FUNCTION_BLOCK TLController (* Composite Function Block Type *)
  (* Standard: 61499-2 *)
  (* Version 0.2, 2003-12-05, JHC, Rockwell Automation, Renamed from NEWCOMPFB. *)
  (* Version 0.1, 2002-01-08, JHC, Rockwell Automation, Added DLY FB as example. *)
  (* Version 0.0, 2000-05-27, JHC, Rockwell Automation *)
  (* Compiler header: package fb.rt.template; *)
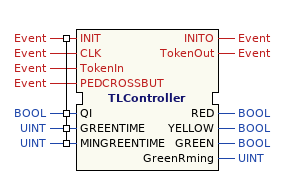
  EVENT_INPUT
    INIT WITH QI, GREENTIME, MINGREENTIME; (* Initialization Request *)
    CLK;
    TokenIn;
    PEDCROSSBUT;
  END_EVENT
  EVENT_OUTPUT
    INITO; (* Initialization Confirm *)
    TokenOut;
  END_EVENT
  VAR_INPUT
    QI : BOOL; (* Input event qualifier *)
    GREENTIME : UINT;
    MINGREENTIME : UINT;
  END_VAR
  VAR_OUTPUT
    RED : BOOL;
    YELLOW : BOOL;
    GREEN : BOOL;
    GreenRming : UINT;
  END_VAR
  FBS
    ButPressCTR : E_CTU(PV := 4);
    Controller : Controller;
    CLOCK : E_CYCLE(DT := t#1s);
    Split1 : E_SPLIT;
  END_FBS
  EVENT_CONNECTIONS
    PEDCROSSBUT TO ButPressCTR.CU;
    Controller.OUTTOKEN TO Split1.EI;
    Split1.EO1 TO TokenOut;
    Split1.EO2 TO CLOCK.STOP;
    INIT TO Controller.INIT;
    INIT TO CLOCK.START;
    TokenIn TO CLOCK.START;
    CLOCK.EO TO Controller.CLK;
  END_CONNECTIONS
  DATA_CONNECTIONS
    Controller.RED TO RED;
    Controller.YELLOW TO YELLOW;
    Controller.GREEN TO GREEN;
    GREENTIME TO Controller.GREENTIME;
    MINGREENTIME TO Controller.MINGREENTIME;
    ButPressCTR.Q TO Controller.PEDCROSS;
  END_CONNECTIONS
END_FUNCTION_BLOCK
